KUKA KRL data list: fri_isir_control.dat

&ACCESS RVO
&REL 59
&COMMENT ISIR-CNRS 2016
&PARAM start_pose = {a1 91.88,a2 112.87,a3 -102.22,a4 6.83,a5 55.73,a6 9.67,e1 -6.27}
&PARAM tool_number = 10
&PARAM TEMPLATE = C:\KRC\Roboter\Template\vorgabe
&PARAM fri_rate_ms = 1.0
&PARAM base_number = 0
&PARAM EDITMASK = *
DEFDAT fri_isir_control PUBLIC

EXT  BAS (BAS_COMMAND  :IN,REAL  :IN )
DECL INT SUCCESS

INT i
DECL GLOBAL BOOL use_rel
DECL GLOBAL INT input_type
DECL FRISTATE ret
REAL fri_rate_ms
INT  tool_number
DECL GLOBAL E6AXIS start_pose
DECL GLOBAL E6AXIS JOINT_CMD
DECL GLOBAL E6POS CART_CMD

ENDDAT
